FUNCTION_BLOCK RT_E_SPLIT (* Split an event to two event chain branches *)
  (* Description: Copyright (c) 2008 ACIN This program and the accompanying materials are made available under the terms of the Eclipse Public License 2.0 which is available at https://www.eclipse.org/legal/epl-2.0/ SPDX-License-Identifier: EPL-2.0 *)
  (* Version 1.0, 2008-07-10, Alois Zoitl, ACIN *)
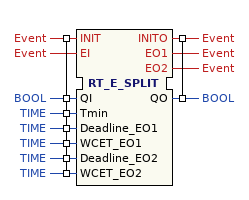
  EVENT_INPUT
    INIT WITH QI, Tmin, Deadline_EO1, WCET_EO1, Deadline_EO2, WCET_EO2;
    EI; (* Input event *)
  END_EVENT
  EVENT_OUTPUT
    INITO WITH QO;
    EO1; (* First output event *)
    EO2; (* Second output event,etc. *)
  END_EVENT
  VAR_INPUT
    QI : BOOL;
    Tmin : TIME;
    Deadline_EO1 : TIME;
    WCET_EO1 : TIME;
    Deadline_EO2 : TIME;
    WCET_EO2 : TIME;
  END_VAR
  VAR_OUTPUT
    QO : BOOL;
  END_VAR
END_FUNCTION_BLOCK
